TYPE
    PLCopenCallInternal :
    STRUCT
        _state : PLCopenCallState;
        _Command : IPLCopenCommand;
        _abort : BOOL;
        _execute : BOOL;
        _break : BOOL;
        _RemoteStatus : PLCopenStatusBase;
        _self : IPLCopenCall;
    END_STRUCT
END_TYPE

(* stored: Version 1.1.0.1
   DUT PLCopenCallInternal: Id {a493e5a4-f6ba-450d-b862-4481c25cddf0} *)
